TYPE ST_HMI_DataSourceCtrl : 
STRUCT
	nActiveMachineIdx: INT;
	nActiveStreamIdx: INT;
	
	bHistorical: BOOL;
	
	//IF Historical
	nActiveRecordIdx: INT;
	
	dtSelectedRangeStart: DCTIMESTRUCT;
	dtSelectedRangeEnd: DCTIMESTRUCT;
	
	bStart: BOOL;
	bCancel: BOOL;
	bPause: BOOL;
	
	bUpdateRecordList: BOOL;
END_STRUCT
END_TYPE

(* stored: Version 1.1.0.1
   DUT ST_HMI_DataSourceCtrl: Id fc9b0aba-b381-4171-b1bd-65342c8e5373 *)
